TYPE ST_DamperRotationMotionConfig :
STRUCT
    fVelocity : LREAL;
    fAcceleration : LREAL;
    fDeceleration : LREAL;
    fPositionTolerance : LREAL;
END_STRUCT
END_TYPE

(* stored: Version 1.1.0.1, ProductVersion 3.1.4026.20
   DUT ST_DamperRotationMotionConfig: Id {5d0aac0c-9f8b-45ad-ad9d-c78dc2d2e025} *)
